PROGRAM A04_StartupWebHMI
VAR
	aStartHMI: ARRAY[1..2] OF NT_StartProcess;
	aPulse: ARRAY[1..2] OF FB_SquareWave;
	aNotRunning:ARRAY[1..2] OF  TON;
	aBusyOnce	:ARRAY[1..2] OF BOOL;

	aWatchdog: ARRAY[1..2] OF TON;
	aLastWatchdogFromHMI	:ARRAY[1..2] OF DINT;
	aWait:ARRAY[1..2] OF BOOL;

	aHMILocalRun :ARRAY[1..2] OF BOOL;
END_VAR

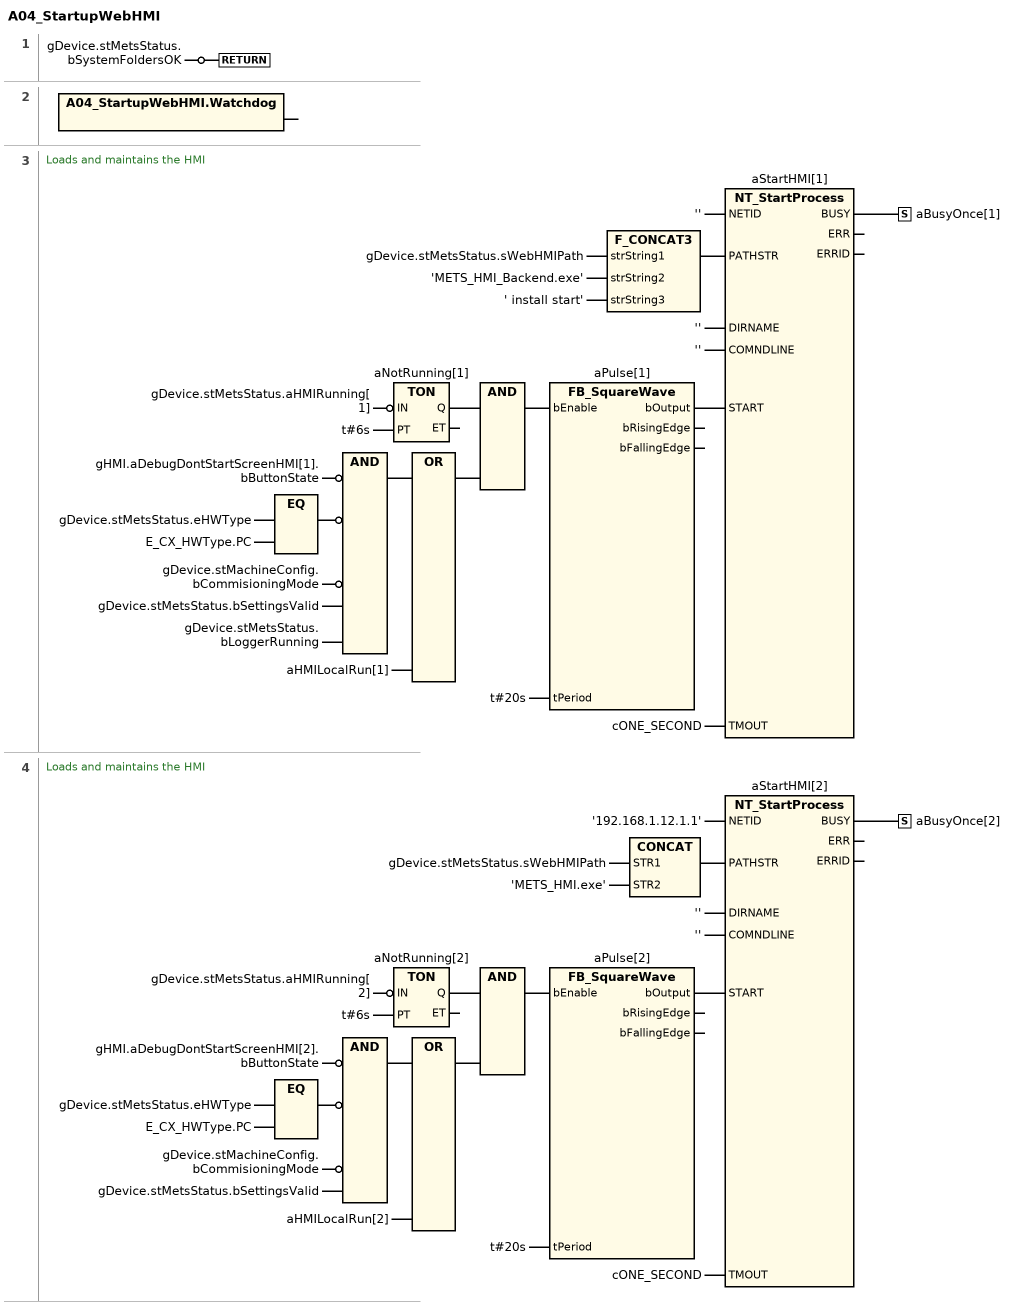
// NETWORK 1
IF NOT gDevice.stMetsStatus.bSystemFoldersOK THEN RETURN; END_IF

// NETWORK 2
A04_StartupWebHMI.Watchdog();

// NETWORK 3
// Loads and maintains the HMI
aNotRunning[1](IN := NOT gDevice.stMetsStatus.aHMIRunning[1], PT := t#6s); // TON
aPulse[1](bEnable := aNotRunning[1].Q AND (NOT gHMI.aDebugDontStartScreenHMI[1].bButtonState AND NOT (gDevice.stMetsStatus.eHWType = E_CX_HWType.PC) AND NOT gDevice.stMachineConfig.bCommisioningMode AND gDevice.stMetsStatus.bSettingsValid AND gDevice.stMetsStatus.bLoggerRunning OR aHMILocalRun[1]), tPeriod := t#20s); // FB_SquareWave
aStartHMI[1](
    NETID := '',
    PATHSTR := F_CONCAT3(strString1 := gDevice.stMetsStatus.sWebHMIPath, strString2 := 'METS_HMI_Backend.exe', strString3 := ' install start'),
    DIRNAME := '',
    COMNDLINE := '',
    START := aPulse[1].bOutput,
    TMOUT := cONE_SECOND); // NT_StartProcess
aBusyOnce[1] S= aStartHMI[1].BUSY;

// NETWORK 4
// Loads and maintains the HMI
aNotRunning[2](IN := NOT gDevice.stMetsStatus.aHMIRunning[2], PT := t#6s); // TON
aPulse[2](bEnable := aNotRunning[2].Q AND (NOT gHMI.aDebugDontStartScreenHMI[2].bButtonState AND NOT (gDevice.stMetsStatus.eHWType = E_CX_HWType.PC) AND NOT gDevice.stMachineConfig.bCommisioningMode AND gDevice.stMetsStatus.bSettingsValid OR aHMILocalRun[2]), tPeriod := t#20s); // FB_SquareWave
aStartHMI[2](
    NETID := '192.168.1.12.1.1',
    PATHSTR := CONCAT(STR1 := gDevice.stMetsStatus.sWebHMIPath, STR2 := 'METS_HMI.exe'),
    DIRNAME := '',
    COMNDLINE := '',
    START := aPulse[2].bOutput,
    TMOUT := cONE_SECOND); // NT_StartProcess
aBusyOnce[2] S= aStartHMI[2].BUSY;

ACTION Watchdog:
(*Watchdog to HMI. HMI closes if PLC stops*)
gHMI.aWatchdogToHMI[1] := gHMI.aWatchdogToHMI[1] + 1;
IF  gHMI.aWatchdogToHMI[1] > 100000 THEN
	gHMI.aWatchdogToHMI[1] := 1;
END_IF

(*Watchdog from HMI - check if running*)
IF aWatchdog[1].Q THEN
	aWait[1] := FALSE;
	IF gHMI.aWatchdogFromHMI[1] <> aLastWatchdogFromHMI[1] THEN
		gDevice.stMetsStatus.aHMIRunning[1] := TRUE;
		aLastWatchdogFromHMI[1] := gHMI.aWatchdogFromHMI[1];
	ELSE
		gDevice.stMetsStatus.aHMIRunning[1] := FALSE;
	END_IF
ELSE
	aWait[1] := TRUE;
END_IF

aWatchdog[1](IN:= aWait[1], PT := t#4000ms);

gDevice.stMetsStatus.aHMIRunning[1] := TRUE;  {warning 'HMI state is overwritten in P01'}

(***********************************************************************************)

(*Watchdog to HMI. HMI closes if PLC stops*)
gHMI.aWatchdogToHMI[2] := gHMI.aWatchdogToHMI[2] + 1;
IF  gHMI.aWatchdogToHMI[2] > 100000 THEN
	gHMI.aWatchdogToHMI[2] := 1;
END_IF

(*Watchdog from HMI - check if running*)
IF aWatchdog[2].Q THEN
	aWait[2] := FALSE;
	IF gHMI.aWatchdogFromHMI[2] <> aLastWatchdogFromHMI[2] THEN
		gDevice.stMetsStatus.aHMIRunning[2] := TRUE;
		aLastWatchdogFromHMI[2] := gHMI.aWatchdogFromHMI[2];
	ELSE
		gDevice.stMetsStatus.aHMIRunning[2] := FALSE;
	END_IF
ELSE
	aWait[2] := TRUE;
END_IF

aWatchdog[2](IN:= aWait[2], PT := t#4000ms);
END_ACTION

END_PROGRAM

(* stored: Version 1.1.0.1
   POU A04_StartupWebHMI: Id {f2a3edc1-242b-47d8-bd15-ccc2f497f607}, SpecialFunc None
   Action Watchdog: Id {4532c039-96a0-4ba6-a583-559cd094941b} *)
